// TIA Portal V20 export
DATA_BLOCK "SP507"   // DB323
// stored: MemoryReserve 100
   VAR
      "PHMI-1 EMERGENCY STOP CH.A" : Bool;
      "PHMI-1 ENABLE SWITCH CH.A" : Bool;
      "PHMI-2 EMERGENCY STOP CH.A" : Bool;
      "PHMI-2 ENABLE SWITCH CH.A" : Bool;
      "PHMI-1 EMERGENCY STOP CH.B" : Bool;
      "PHMI-1 ENABLE SWITCH CH.B" : Bool;
      "PHMI-2 EMERGENCY STOP CH.B" : Bool;
      "PHMI-2 ENABLE SWITCH CH.B" : Bool;
   END_VAR
BEGIN
END_DATA_BLOCK
